FUNCTION_BLOCK JSON_DESERIALIZER (* Composite FB wrapping other FBs *)
  (* Standard: 61499-2 *)
  (* Version 1.0, 2023-04-20, valentinnodan *)
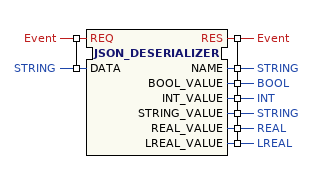
  EVENT_INPUT
    REQ WITH DATA; (* Normal Execution Request *)
  END_EVENT
  EVENT_OUTPUT
    RES WITH BOOL_VALUE, INT_VALUE, STRING_VALUE, REAL_VALUE, LREAL_VALUE, NAME; (* Execution Confirmation *)
  END_EVENT
  VAR_INPUT
    DATA : STRING; (* Input event qualifier *)
  END_VAR
  VAR_OUTPUT
    NAME : STRING;
    BOOL_VALUE : BOOL; (* Output event qualifier *)
    INT_VALUE : INT;
    STRING_VALUE : STRING;
    REAL_VALUE : REAL;
    LREAL_VALUE : LREAL;
  END_VAR
  FBS
    TYPE_DETECTOR : TYPE_DETECTOR;
    JSON_PARSER : JSON_PARSER;
    F_STRING_TO_BOOL : F_STRING_TO_BOOL;
    F_STRING_TO_INT : F_STRING_TO_INT;
    F_STRING_TO_REAL : F_STRING_TO_REAL;
    F_STRING_TO_LREAL : F_STRING_TO_LREAL;
  END_FBS
  EVENT_CONNECTIONS
    REQ TO JSON_PARSER.REQ;
    JSON_PARSER.RES TO TYPE_DETECTOR.REQ;
    TYPE_DETECTOR.IS_BOOL TO F_STRING_TO_BOOL.REQ;
    F_STRING_TO_BOOL.CNF TO RES;
    TYPE_DETECTOR.IS_INT TO F_STRING_TO_INT.REQ;
    TYPE_DETECTOR.IS_REAL TO F_STRING_TO_REAL.REQ;
    TYPE_DETECTOR.IS_LREAL TO F_STRING_TO_LREAL.REQ;
    F_STRING_TO_INT.CNF TO RES;
    F_STRING_TO_REAL.CNF TO RES;
    F_STRING_TO_LREAL.CNF TO RES;
    TYPE_DETECTOR.IS_STRING TO RES;
  END_CONNECTIONS
  DATA_CONNECTIONS
    DATA TO JSON_PARSER.DATA;
    JSON_PARSER.TYPE TO TYPE_DETECTOR.TYPE_NAME;
    JSON_PARSER.VALUE TO F_STRING_TO_BOOL.IN;
    JSON_PARSER.VALUE TO F_STRING_TO_INT.IN;
    F_STRING_TO_BOOL.OUT TO BOOL_VALUE;
    JSON_PARSER.NAME TO NAME;
    JSON_PARSER.VALUE TO F_STRING_TO_REAL.IN;
    JSON_PARSER.VALUE TO F_STRING_TO_LREAL.IN;
    F_STRING_TO_INT.OUT TO INT_VALUE;
    F_STRING_TO_REAL.OUT TO REAL_VALUE;
    F_STRING_TO_LREAL.OUT TO LREAL_VALUE;
    JSON_PARSER.VALUE TO STRING_VALUE;
  END_CONNECTIONS
END_FUNCTION_BLOCK
